INTERFACE I_State

PROPERTY P_State : INT
GET
END_GET
END_PROPERTY

END_INTERFACE

(* stored: Version 1.1.0.1
   Itf I_State: Id {c9f25642-45e6-46ba-9b60-272faa0dde20}
   Property P_State: Id {d32fab83-0766-4ce0-8cc8-38f2daa7745e}
   Get Get: Id {58c5b2c3-ef63-4a33-a60e-64381cd02dc7} *)
